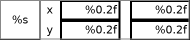
VISUALIZATION _VISU_PlacementXY_puc  // 190x40
VAR_IN_OUT
	mInst : ST_CORRECTION_POINT;
  aName : STRING;
  bSelected : BOOL;
  bSelect : BOOL;
END_VAR
    Rectangle (40,0 20x20), "x"
    Rectangle (40,20 20x20), "y"
    Rectangle (0,0 40x40), "%s", text variable: aName, colour toggle: bSelected
        toggle bSelect
    Rectangle (60,0 60x20), "%0.2f", tooltip "reference", text variable: mInst.posx
        OnMouseClick: write the text variable via Default
    Rectangle (60,20 60x20), "%0.2f", tooltip "reference", text variable: mInst.posy
        OnMouseClick: write the text variable via Default
    Rectangle (130,0 60x20), "%0.2f", tooltip "correction relative", text variable: mInst.x
        OnMouseClick: write the text variable via Default
    Rectangle (130,20 60x20), "%0.2f", tooltip "correction relative", text variable: mInst.y
        OnMouseClick: write the text variable via Default
END_VISUALIZATION

(* stored: Version 1.1.0.1, ProductVersion 3.1.4024.11
   Visu _VISU_PlacementXY_puc: Id {bce341c7-f186-482a-abdc-51c84728ad03} *)
